Staubli VAL3: MSGBOX.pgx

public program msgBox(string x_sMessage, num x_nBoxWidth, string x_sChoice, num& x_nSelectedFKey[])
  local num l_i
  local num l_nKeyPressed
  local num l_nError
  local num l_nRow
  local num l_nCol
begin
  // This program displays a message box on the MCP
  // and wait for the answer of the user.
  //
  // Input param
  // x_sMessage    : Message to display
  // x_nBoxWidth   : width of the message box to display
  // x_sChoice     : Different choices for the user (typically YES  NO  CANCEL)
  //
  // Output param
  // x_nSelectedFKey  : Number of the functio n key pressed by user
  //        range is 1 to 8
  //
  // Created 23-02-05                           C.CURRIVAND
  //------------------------------------------------------------------
  //
  // Set default width if parameter is not consistent
  if x_nBoxWidth<=0
    x_nBoxWidth=5
  endIf
  l_nRow=3
  //
  // Format the message to display (result is array of string called sWrkString[])
  // BoxWidth may be adjusted if one string is longer than boxWidth
  call setString(x_sMessage,x_nBoxWidth,l_nError)
  l_nCol=roundDown((40-x_nBoxWidth)/2)
  //
  // display message Box
  nTxtBoxCol=l_nCol
  nTxtBoxRow=l_nRow
  nTxtBoxWidth=x_nBoxWidth-2
  call msgBoxDisplay(x_nBoxWidth)
  //
  // Erase last line of screen
  call clear(0,13)
  call displayMenu(x_sChoice)
  do
    call GetFKey(x_sChoice,l_nKeyPressed)
    delay(0)
  until (l_nKeyPressed>=1) and (l_nKeyPressed<=8)
  x_nSelectedFKey=l_nKeyPressed
end
